# EPICS autosave request: trunk/stdApp/Db/femto.req
$(P)$(H)$(F)debug
$(P)$(H)$(F)gain
$(P)$(H)$(F)gainidx
$(P)$(H)$(F)femtodesc
